SUBAPPLICATION Uebung_010a (* SoftKey_F1/_F2 auf DigitalOutput_Q1/_Q2 *)
  (* Standard: 61499-2 *)
  (* Version 1.0, 2023-10-23, franz *)
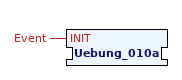
  EVENT_INPUT
    INIT;
  END_EVENT
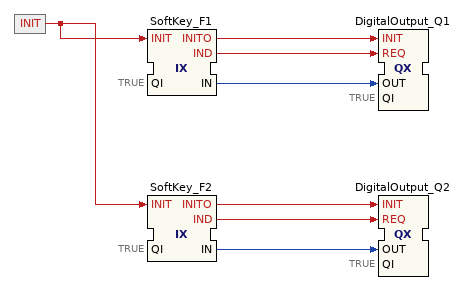
  FBS
    DigitalOutput_Q1 : QX(QI := TRUE);
    SoftKey_F1 : IX(QI := TRUE);
    SoftKey_F2 : IX(QI := TRUE);
    DigitalOutput_Q2 : QX(QI := TRUE);
  END_FBS
  EVENT_CONNECTIONS
    INIT TO SoftKey_F1.INIT;
    SoftKey_F1.INITO TO DigitalOutput_Q1.INIT;
    SoftKey_F1.IND TO DigitalOutput_Q1.REQ;
    SoftKey_F2.INITO TO DigitalOutput_Q2.INIT;
    SoftKey_F2.IND TO DigitalOutput_Q2.REQ;
    INIT TO SoftKey_F2.INIT;
  END_CONNECTIONS
  DATA_CONNECTIONS
    SoftKey_F1.IN TO DigitalOutput_Q1.OUT;
    SoftKey_F2.IN TO DigitalOutput_Q2.OUT;
  END_CONNECTIONS
END_SUBAPPLICATION
